(*

.. <legal notes>

legal notes
=================
| SPDX-FileCopyrightText: © 2025 Oleksandr Tiutyk <trofimich@gmail.com>
| SPDX-License-Identifier: LGPL-3.0-only
| For details check: LGPL-3.0-only_

.. _LGPL-3.0-only: https://www.gnu.org/licenses/lgpl-3.0.en.html

.. </legal notes>

*)

INTERFACE IEnumerator EXTENDS IObject

// Shows curent collection element
PROPERTY ABSTRACT Current : REFERENCE TO GENERIC_VALUE
GET
END_GET
END_PROPERTY

// Moves Current pointer to next collection element
METHOD MoveNext : BOOL
END_METHOD

// Sets the enumerator to its initial position, which is before the first element in the collection
METHOD Reset
END_METHOD

END_INTERFACE

(* stored: Version 1.1.0.1
   Itf IEnumerator: Id {459ae103-383b-4a03-9f68-f28a3cccf087}
   Property Current: Id {6246802f-40aa-48e9-b7fb-975da88bd2b5}
   Get Get: Id {cc639373-80a5-4044-8578-7fe884c3c23a}
   Method MoveNext: Id {c36c1566-0815-4b50-a29c-445adbeb3671}
   Method Reset: Id {959ae268-37f4-4623-916b-c48b391e2a9b} *)
